(* IEC 61131-3 sources: CodesysTest/alpha/export/FBs/Components/BagOpenFingersWithSensorsFB.pou, 1 file *)

(* ---- BagOpenFingersWithSensorsFB.pou.st ---- *)
(*#-#-#-#-#-#-#-#-#-#---Declaration---#-#-#-#-#-#-#-#-#-#-#-#-#*)

FUNCTION_BLOCK BagOpenFingersWithSensorsFB EXTENDS BagOpenFingersFB
VAR_INPUT
	rightFingerBagPresent : BOOL;
	leftFingerBagPreset : BOOL;
END_VAR
VAR_IN_OUT
	bagFailedToGrabBothFingersCount : UDINT; // Both Fingers failed to grab bag
	bagFailedToGrabRightFingerCount : UDINT; // Right Bag Open Finger Failed to Grab Bag
	bagFailedToGrabLeftFingerCount : UDINT; // Left Bag Open Finger Failed to Grab Bag
	successfulBagOpenCount : UDINT;			// Successful Bag Open Count
END_VAR
VAR_OUTPUT

END_VAR
(*#-#-#-#-#-#-#-#-#-#---Implementation---#-#-#-#-#-#-#-#-#-#-#-#-#*)

SUPER^();
